FUNCTION_BLOCK FB_ActivateAction EXTENDS TcBase.FB_Action
VAR
    _bActivated: BOOL;
END_VAR

METHOD  Execute
VAR_INPUT
    ipObject: I_Object;
END_VAR
VAR
    p: POINTER TO FB_ActionTestObject;
END_VAR
__QUERYPOINTER(ipObject, p);

IF p <> 0 THEN
    p^.Activate(THIS^._bActivated);
END_IF
END_METHOD

METHOD Inputs : TcBase.I_Action
VAR_INPUT
    bActivate: BOOL;
END_VAR
Inputs := THIS^;
THIS^._bActivated := bActivate;
END_METHOD

END_FUNCTION_BLOCK

(* stored: Version 1.1.0.1, ProductVersion 3.1.4024.12
   POU FB_ActivateAction: Id {7e404be6-fc8b-4051-988f-7033ffb613a4}, SpecialFunc None
   Method Execute: Id {fc2eff42-265e-4bd3-b080-5d930c8ab5c6}
   Method Inputs: Id {e6bc8e59-7bf0-479b-a73a-f39b72e7c2f9} *)
